PROGRAM KrAxis
VAR
//	KR_Axis_V2_Carriage: KR_Achse_v2; //set up control box, BUT NOT REAL CONTROL
//	Adapter_Carriage: FB_AdapterSI6; // adapter needed to make sure the information is passed correctly
	
	RefTrigger: BOOL; // trigger from a sensor to mark the referance point
	CycleTime: REAL := 0.001; // cycle time of the block. MAKE SURE ITS IN THE 1MS zone
	MMpMotorROT :LREAL := 100;  // mm per motor rotation. used in planar travel. basically its how big the moving wheel is. 
//	FollowErrorVelCorrection: LREAL := 1; // german only tool!!!! a follow error correction that acts with the drive. wikipedia "KR FAKTOR". VERY useful!
//	StoppingWindow: LREAL := 1; // the window the drive has to stop close to the target and designate its self in the right spot
//	DriveInverted: BOOL; // activate if there is wrong wiring on the drive. NOT for going BACKWARDS!!!!
		
	EncoderFactorMMpINC: LREAL := 0.000095; //standard encoder factor for mm per inc. very important to get this right. take mmpMotorRot / 1048576
	
	RefSearchVEL: LREAL := 50; //Velocity of drive when it is searching for the referance.
	RefFoundVEL: LREAL := 50; //used in the 'steping away' move from the sensor after it is found. NOT FOR REGULAR USE
	
//	FollowErrorVelLimit: LREAL := 15;// the top speed KV2 can move up. larger mass makes it bigger
//	FollowErrorVelGAIN: REAL := 0; // the gain the KV velocity will use to try and keep up. 0 is good. large mass makes it bigger
	
	SetTheoreticPos: BOOL; // activates a theortical postion for the drive to and simulate 
	TheoreticPos: LREAL; // the theoretical target position
	TheoreticVelo: LREAL; // the speed it uses to get to this theoretical position.
	EncoderType: BOOL; // 1 for incremental, 0 for absolute
	
//	MiddleEncoderValue: LREAL; // the middle of between the max and min vlaue. this will watch for an roll overs 
	Sim: BOOL; // cause a simulation for the drive to react but the motor does not spin. use this same tag for all FB sim modes!!!!
	JumpErrorWindow: REAL; // causes an error if something happens between two cycles. like the inverter tell the drive to move too fast.

	
//	NominalRotations: REAL := 3000;  // labeled as "nN" on the motor. make sure its not a '.' vs a ',' (should be in the 1000, depending on motor) 
	MaxEncoderIncriments: DWORD := 1048576; // almost always 1048576!!!! this is the multiplied factor of the max encoder counts
	  
	
(* ##### INITIAL DRIVE SETUP ##### *)

//Carriage
	KR_Axis_V2_Carriage: KR_Achse_v2; //set up control box, BUT NOT REAL CONTROL
	Adapter_Carriage: FB_AdapterSI6; // adapter needed to make sure the information is passed correctly

	CRG_FollowErrorVelCorrection: LREAL := 15; // german only tool!!!! a follow error correction that acts with the drive. wikipedia "KR FAKTOR". VERY useful!
	CRG_StoppingWindow: LREAL := 1; // the window the drive has to stop close to the target and designate its self in the right spot
	CRG_DriveInverted: BOOL; // activate if there is wrong wiring on the drive. NOT for going BACKWARDS!!!!
	CRG_FollowErrorVelLimit: LREAL := 600;// the top speed KV2 can move up. larger mass makes it bigger
	CRG_FollowErrorVelGAIN: REAL := 0; // the gain the KV velocity will use to try and keep up. 0 is good. large mass makes it bigger
	CRG_MiddleEncoderValue: LREAL := 20744.82692; // the middle of between the max and min vlaue. this will watch for an roll overs 
	CRG_NominalRotations: REAL := 6000;  // labeled as "nN" on the motor. make sure its not a '.' vs a ',' (should be in the 1000, depending on motor) 

//Turret
	KR_Axis_V2_Turret: KR_Achse_v2; //set up control box, BUT NOT REAL CONTROL
	Adapter_Turret: FB_AdapterSI6; // adapter needed to make sure the information is passed correctly

	TRT_FollowErrorVelCorrection: LREAL := 15; // german only tool!!!! a follow error correction that acts with the drive. wikipedia "KR FAKTOR". VERY useful!
	TRT_StoppingWindow: LREAL := 0.1; // the window the drive has to stop close to the target and designate its self in the right spot
	TRT_DriveInverted: BOOL; // activate if there is wrong wiring on the drive. NOT for going BACKWARDS!!!!
	TRT_FollowErrorVelLimit: LREAL := 300;// the top speed KV2 can move up. larger mass makes it bigger
	TRT_FollowErrorVelGAIN: REAL := 0; // the gain the KV velocity will use to try and keep up. 0 is good. large mass makes it bigger
	TRT_MiddleEncoderValue: LREAL := 1296.282433; // the middle of between the max and min vlaue. this will watch for an roll overs 
	TRT_NominalRotations: REAL := 3000;  // labeled as "nN" on the motor. make sure its not a '.' vs a ',' (should be in the 1000, depending on motor) 

	//CrossCut
	KR_Axis_V2_CrossCut: KR_Achse_v2; //set up control box, BUT NOT REAL CONTROL
	Adapter_CrossCut: FB_AdapterSI6; // adapter needed to make sure the information is passed correctly

	CRC_FollowErrorVelCorrection: LREAL := 15; // german only tool!!!! a follow error correction that acts with the drive. wikipedia "KR FAKTOR". VERY useful!
	CRC_StoppingWindow: LREAL := 1; // the window the drive has to stop close to the target and designate its self in the right spot
	CRC_DriveInverted: BOOL; // activate if there is wrong wiring on the drive. NOT for going BACKWARDS!!!!
	CRC_FollowErrorVelLimit: LREAL := 600;// the top speed KV2 can move up. larger mass makes it bigger
	CRC_FollowErrorVelGAIN: REAL := 0; // the gain the KV velocity will use to try and keep up. 0 is good. large mass makes it bigger
	CRC_MiddleEncoderValue: LREAL := 7838.457838; // the middle of between the max and min vlaue. this will watch for an roll overs 
	CRC_NominalRotations: REAL := 6000;  // labeled as "nN" on the motor. make sure its not a '.' vs a ',' (should be in the 1000, depending on motor) 

//XDrive
	KR_Axis_V2_XDrive: KR_Achse_v2; //set up control box, BUT NOT REAL CONTROL
	Adapter_XDrive: FB_AdapterSI6; // adapter needed to make sure the information is passed correctly

	XDR_FollowErrorVelCorrection: LREAL := 15; // german only tool!!!! a follow error correction that acts with the drive. wikipedia "KR FAKTOR". VERY useful!
	XDR_StoppingWindow: LREAL := 1; // the window the drive has to stop close to the target and designate its self in the right spot
	XDR_DriveInverted: BOOL; // activate if there is wrong wiring on the drive. NOT for going BACKWARDS!!!!
	XDR_FollowErrorVelLimit: LREAL := 300;// the top speed KV2 can move up. larger mass makes it bigger
	XDR_FollowErrorVelGAIN: REAL := 0; // the gain the KV velocity will use to try and keep up. 0 is good. large mass makes it bigger
	XDR_MiddleEncoderValue: LREAL := 41225.1069; // the middle of between the max and min vlaue. this will watch for an roll overs 
	XDR_NominalRotations: REAL := 3000;  // labeled as "nN" on the motor. make sure its not a '.' vs a ',' (should be in the 1000, depending on motor) 

//Z1
	KR_Axis_V2_Z1: KR_Achse_v2; //set up control box, BUT NOT REAL CONTROL
	Adapter_Z1: FB_AdapterSI6; // adapter needed to make sure the information is passed correctly

	Z1_FollowErrorVelCorrection: LREAL := 15; // german only tool!!!! a follow error correction that acts with the drive. wikipedia "KR FAKTOR". VERY useful!
	Z1_StoppingWindow: LREAL := 1; // the window the drive has to stop close to the target and designate its self in the right spot
	Z1_DriveInverted: BOOL; // activate if there is wrong wiring on the drive. NOT for going BACKWARDS!!!!
	Z1_FollowErrorVelLimit: LREAL := 300;// the top speed KV2 can move up. larger mass makes it bigger
	Z1_FollowErrorVelGAIN: REAL := 0; // the gain the KV velocity will use to try and keep up. 0 is good. large mass makes it bigger
	Z1_MiddleEncoderValue: LREAL := 0; // the middle of between the max and min vlaue. this will watch for an roll overs 
	Z1_NominalRotations: REAL := 3000;  // labeled as "nN" on the motor. make sure its not a '.' vs a ',' (should be in the 1000, depending on motor) 

//Z2
	KR_Axis_V2_Z2: KR_Achse_v2; //set up control box, BUT NOT REAL CONTROL
	Adapter_Z2: FB_AdapterSI6; // adapter needed to make sure the information is passed correctly

	Z2_FollowErrorVelCorrection: LREAL := 15; // german only tool!!!! a follow error correction that acts with the drive. wikipedia "KR FAKTOR". VERY useful!
	Z2_StoppingWindow: LREAL := 1; // the window the drive has to stop close to the target and designate its self in the right spot
	Z2_DriveInverted: BOOL; // activate if there is wrong wiring on the drive. NOT for going BACKWARDS!!!!
	Z2_FollowErrorVelLimit: LREAL := 300;// the top speed KV2 can move up. larger mass makes it bigger
	Z2_FollowErrorVelGAIN: REAL := 0; // the gain the KV velocity will use to try and keep up. 0 is good. large mass makes it bigger
	Z2_MiddleEncoderValue: LREAL := 0; // the middle of between the max and min vlaue. this will watch for an roll overs 
	Z2_NominalRotations: REAL := 3000;  // labeled as "nN" on the motor. make sure its not a '.' vs a ',' (should be in the 1000, depending on motor) 

	ZaxisRefTrigger: BOOL;
	
END_VAR

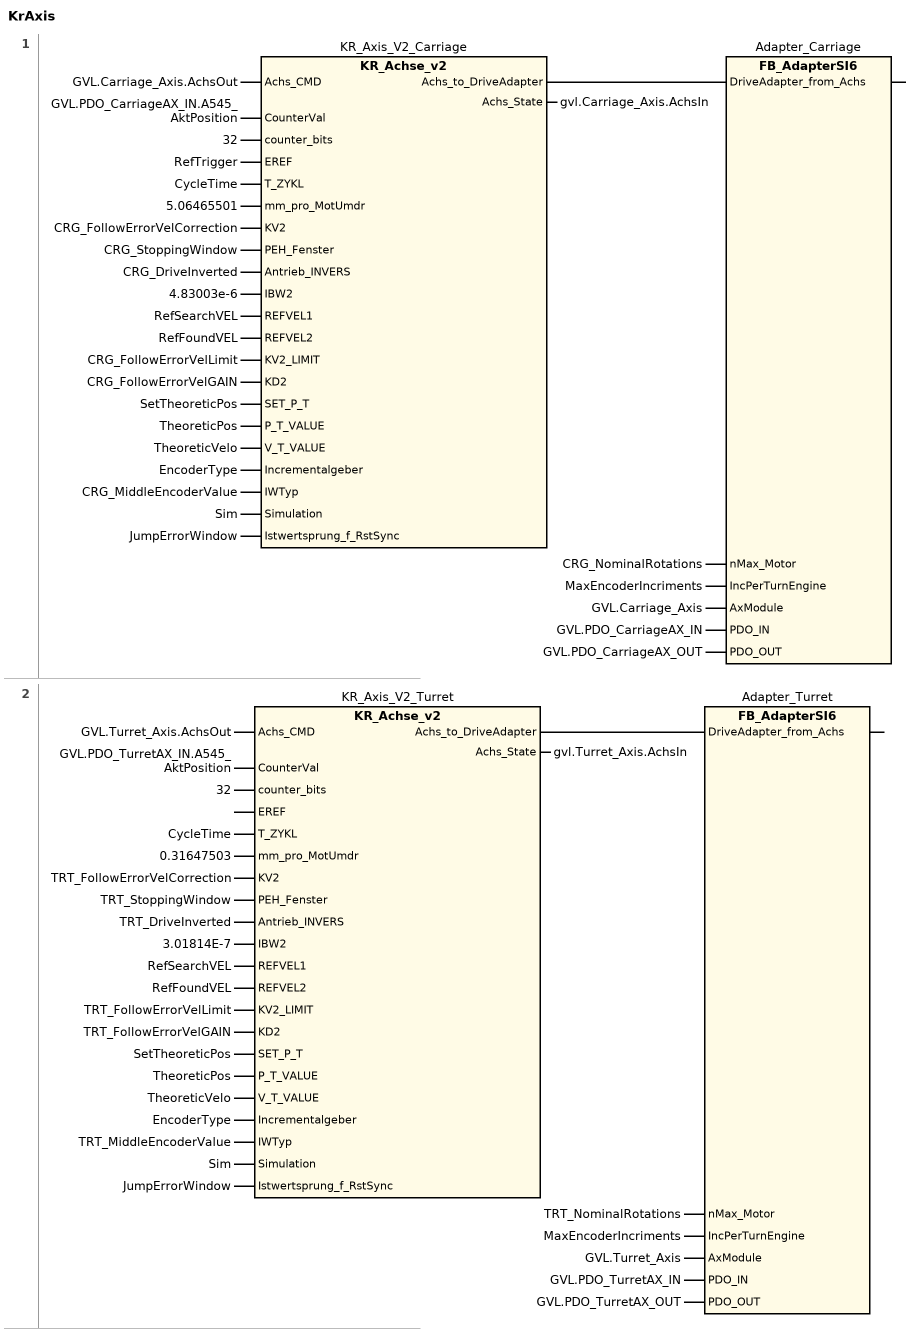
// NETWORK 1
KR_Axis_V2_Carriage(
    Achs_CMD := GVL.Carriage_Axis.AchsOut,
    CounterVal := GVL.PDO_CarriageAX_IN.A545_AktPosition,
    counter_bits := 32,
    EREF := RefTrigger,
    T_ZYKL := CycleTime,
    mm_pro_MotUmdr := 5.06465501,
    KV2 := CRG_FollowErrorVelCorrection,
    PEH_Fenster := CRG_StoppingWindow,
    Antrieb_INVERS := CRG_DriveInverted,
    IBW2 := 4.83003e-6,
    REFVEL1 := RefSearchVEL,
    REFVEL2 := RefFoundVEL,
    KV2_LIMIT := CRG_FollowErrorVelLimit,
    KD2 := CRG_FollowErrorVelGAIN,
    SET_P_T := SetTheoreticPos,
    P_T_VALUE := TheoreticPos,
    V_T_VALUE := TheoreticVelo,
    Incrementalgeber := EncoderType,
    IWTyp := CRG_MiddleEncoderValue,
    Simulation := Sim,
    Istwertsprung_f_RstSync := JumpErrorWindow,
    Achs_State => gvl.Carriage_Axis.AchsIn); // KR_Achse_v2
Adapter_Carriage(
    DriveAdapter_from_Achs := KR_Axis_V2_Carriage.Achs_to_DriveAdapter,
    nMax_Motor := CRG_NominalRotations,
    IncPerTurnEngine := MaxEncoderIncriments,
    AxModule := GVL.Carriage_Axis,
    PDO_IN := GVL.PDO_CarriageAX_IN,
    PDO_OUT := GVL.PDO_CarriageAX_OUT); // FB_AdapterSI6

// NETWORK 2
KR_Axis_V2_Turret(
    Achs_CMD := GVL.Turret_Axis.AchsOut,
    CounterVal := GVL.PDO_TurretAX_IN.A545_AktPosition,
    counter_bits := 32,
    T_ZYKL := CycleTime,
    mm_pro_MotUmdr := 0.31647503,
    KV2 := TRT_FollowErrorVelCorrection,
    PEH_Fenster := TRT_StoppingWindow,
    Antrieb_INVERS := TRT_DriveInverted,
    IBW2 := 3.01814E-7,
    REFVEL1 := RefSearchVEL,
    REFVEL2 := RefFoundVEL,
    KV2_LIMIT := TRT_FollowErrorVelLimit,
    KD2 := TRT_FollowErrorVelGAIN,
    SET_P_T := SetTheoreticPos,
    P_T_VALUE := TheoreticPos,
    V_T_VALUE := TheoreticVelo,
    Incrementalgeber := EncoderType,
    IWTyp := TRT_MiddleEncoderValue,
    Simulation := Sim,
    Istwertsprung_f_RstSync := JumpErrorWindow,
    Achs_State => gvl.Turret_Axis.AchsIn); // KR_Achse_v2
Adapter_Turret(
    DriveAdapter_from_Achs := KR_Axis_V2_Turret.Achs_to_DriveAdapter,
    nMax_Motor := TRT_NominalRotations,
    IncPerTurnEngine := MaxEncoderIncriments,
    AxModule := GVL.Turret_Axis,
    PDO_IN := GVL.PDO_TurretAX_IN,
    PDO_OUT := GVL.PDO_TurretAX_OUT); // FB_AdapterSI6

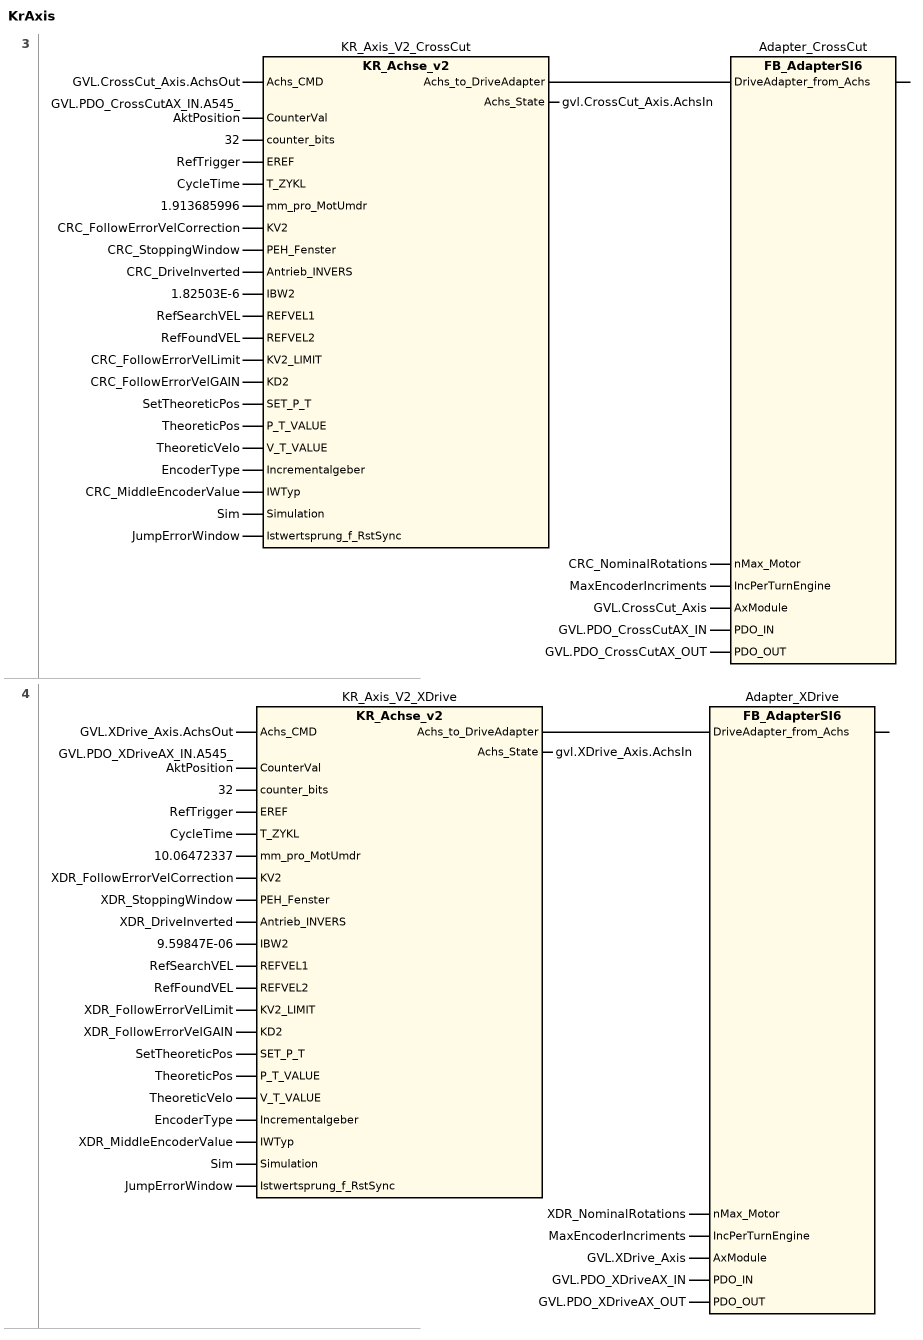
// NETWORK 3
KR_Axis_V2_CrossCut(
    Achs_CMD := GVL.CrossCut_Axis.AchsOut,
    CounterVal := GVL.PDO_CrossCutAX_IN.A545_AktPosition,
    counter_bits := 32,
    EREF := RefTrigger,
    T_ZYKL := CycleTime,
    mm_pro_MotUmdr := 1.913685996,
    KV2 := CRC_FollowErrorVelCorrection,
    PEH_Fenster := CRC_StoppingWindow,
    Antrieb_INVERS := CRC_DriveInverted,
    IBW2 := 1.82503E-6,
    REFVEL1 := RefSearchVEL,
    REFVEL2 := RefFoundVEL,
    KV2_LIMIT := CRC_FollowErrorVelLimit,
    KD2 := CRC_FollowErrorVelGAIN,
    SET_P_T := SetTheoreticPos,
    P_T_VALUE := TheoreticPos,
    V_T_VALUE := TheoreticVelo,
    Incrementalgeber := EncoderType,
    IWTyp := CRC_MiddleEncoderValue,
    Simulation := Sim,
    Istwertsprung_f_RstSync := JumpErrorWindow,
    Achs_State => gvl.CrossCut_Axis.AchsIn); // KR_Achse_v2
Adapter_CrossCut(
    DriveAdapter_from_Achs := KR_Axis_V2_CrossCut.Achs_to_DriveAdapter,
    nMax_Motor := CRC_NominalRotations,
    IncPerTurnEngine := MaxEncoderIncriments,
    AxModule := GVL.CrossCut_Axis,
    PDO_IN := GVL.PDO_CrossCutAX_IN,
    PDO_OUT := GVL.PDO_CrossCutAX_OUT); // FB_AdapterSI6

// NETWORK 4
KR_Axis_V2_XDrive(
    Achs_CMD := GVL.XDrive_Axis.AchsOut,
    CounterVal := GVL.PDO_XDriveAX_IN.A545_AktPosition,
    counter_bits := 32,
    EREF := RefTrigger,
    T_ZYKL := CycleTime,
    mm_pro_MotUmdr := 10.06472337,
    KV2 := XDR_FollowErrorVelCorrection,
    PEH_Fenster := XDR_StoppingWindow,
    Antrieb_INVERS := XDR_DriveInverted,
    IBW2 := 9.59847E-06,
    REFVEL1 := RefSearchVEL,
    REFVEL2 := RefFoundVEL,
    KV2_LIMIT := XDR_FollowErrorVelLimit,
    KD2 := XDR_FollowErrorVelGAIN,
    SET_P_T := SetTheoreticPos,
    P_T_VALUE := TheoreticPos,
    V_T_VALUE := TheoreticVelo,
    Incrementalgeber := EncoderType,
    IWTyp := XDR_MiddleEncoderValue,
    Simulation := Sim,
    Istwertsprung_f_RstSync := JumpErrorWindow,
    Achs_State => gvl.XDrive_Axis.AchsIn); // KR_Achse_v2
Adapter_XDrive(
    DriveAdapter_from_Achs := KR_Axis_V2_XDrive.Achs_to_DriveAdapter,
    nMax_Motor := XDR_NominalRotations,
    IncPerTurnEngine := MaxEncoderIncriments,
    AxModule := GVL.XDrive_Axis,
    PDO_IN := GVL.PDO_XDriveAX_IN,
    PDO_OUT := GVL.PDO_XDriveAX_OUT); // FB_AdapterSI6

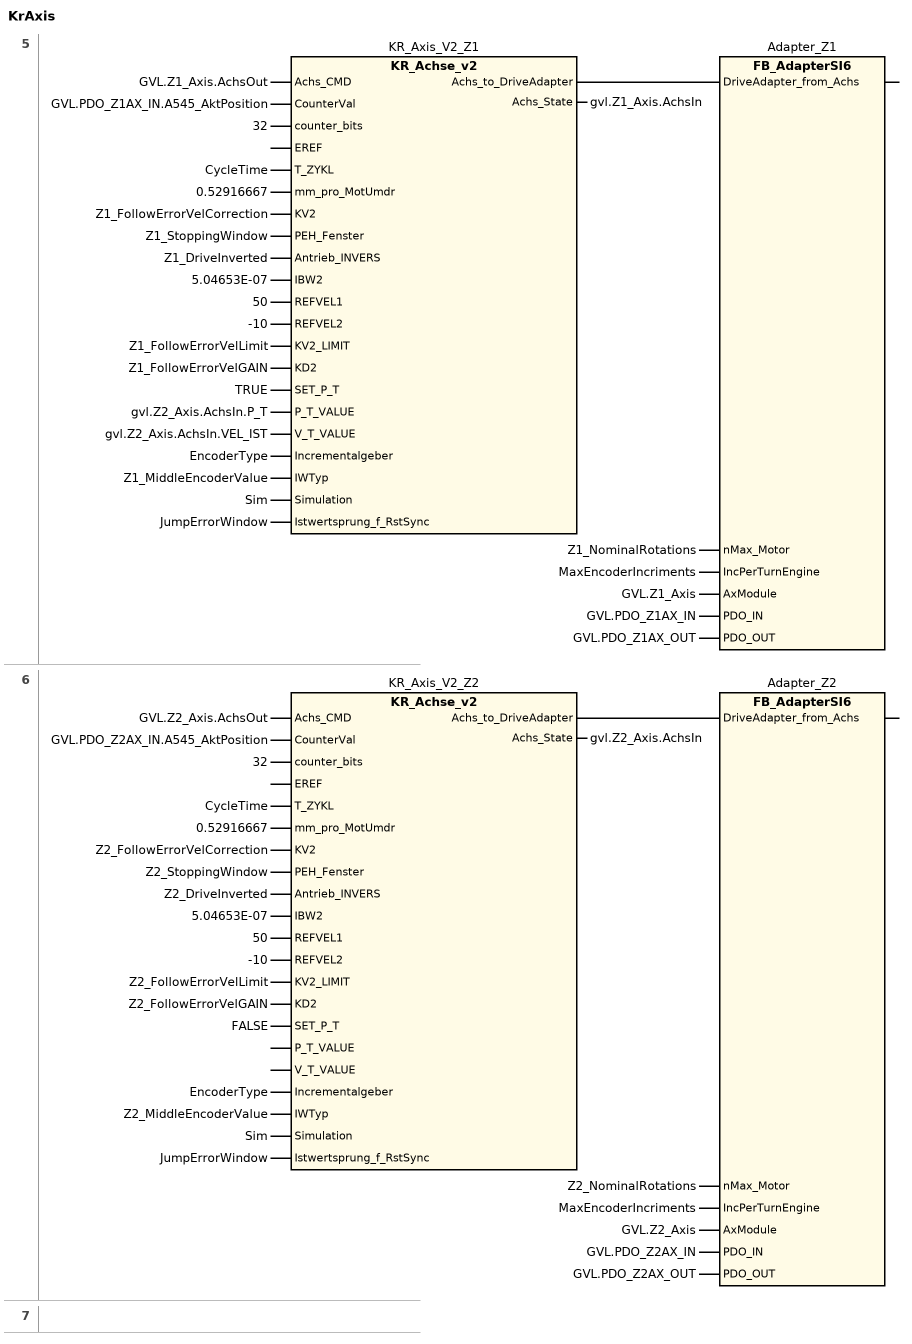
// NETWORK 5
KR_Axis_V2_Z1(
    Achs_CMD := GVL.Z1_Axis.AchsOut,
    CounterVal := GVL.PDO_Z1AX_IN.A545_AktPosition,
    counter_bits := 32,
    T_ZYKL := CycleTime,
    mm_pro_MotUmdr := 0.52916667,
    KV2 := Z1_FollowErrorVelCorrection,
    PEH_Fenster := Z1_StoppingWindow,
    Antrieb_INVERS := Z1_DriveInverted,
    IBW2 := 5.04653E-07,
    REFVEL1 := 50,
    REFVEL2 := -10,
    KV2_LIMIT := Z1_FollowErrorVelLimit,
    KD2 := Z1_FollowErrorVelGAIN,
    SET_P_T := TRUE,
    P_T_VALUE := gvl.Z2_Axis.AchsIn.P_T,
    V_T_VALUE := gvl.Z2_Axis.AchsIn.VEL_IST,
    Incrementalgeber := EncoderType,
    IWTyp := Z1_MiddleEncoderValue,
    Simulation := Sim,
    Istwertsprung_f_RstSync := JumpErrorWindow,
    Achs_State => gvl.Z1_Axis.AchsIn); // KR_Achse_v2
Adapter_Z1(
    DriveAdapter_from_Achs := KR_Axis_V2_Z1.Achs_to_DriveAdapter,
    nMax_Motor := Z1_NominalRotations,
    IncPerTurnEngine := MaxEncoderIncriments,
    AxModule := GVL.Z1_Axis,
    PDO_IN := GVL.PDO_Z1AX_IN,
    PDO_OUT := GVL.PDO_Z1AX_OUT); // FB_AdapterSI6

// NETWORK 6
KR_Axis_V2_Z2(
    Achs_CMD := GVL.Z2_Axis.AchsOut,
    CounterVal := GVL.PDO_Z2AX_IN.A545_AktPosition,
    counter_bits := 32,
    T_ZYKL := CycleTime,
    mm_pro_MotUmdr := 0.52916667,
    KV2 := Z2_FollowErrorVelCorrection,
    PEH_Fenster := Z2_StoppingWindow,
    Antrieb_INVERS := Z2_DriveInverted,
    IBW2 := 5.04653E-07,
    REFVEL1 := 50,
    REFVEL2 := -10,
    KV2_LIMIT := Z2_FollowErrorVelLimit,
    KD2 := Z2_FollowErrorVelGAIN,
    SET_P_T := FALSE,
    Incrementalgeber := EncoderType,
    IWTyp := Z2_MiddleEncoderValue,
    Simulation := Sim,
    Istwertsprung_f_RstSync := JumpErrorWindow,
    Achs_State => gvl.Z2_Axis.AchsIn); // KR_Achse_v2
Adapter_Z2(
    DriveAdapter_from_Achs := KR_Axis_V2_Z2.Achs_to_DriveAdapter,
    nMax_Motor := Z2_NominalRotations,
    IncPerTurnEngine := MaxEncoderIncriments,
    AxModule := GVL.Z2_Axis,
    PDO_IN := GVL.PDO_Z2AX_IN,
    PDO_OUT := GVL.PDO_Z2AX_OUT); // FB_AdapterSI6

// NETWORK 7

END_PROGRAM

(* stored: Version 1.1.0.1, ProductVersion 3.1.4024.15
   POU KrAxis: Id {1a1067ba-3531-4527-95c4-b5f18a11280c}, SpecialFunc None *)
